TYPE ST_ProbesSettings :
STRUCT
	
	anDistanceCalibrationBlock			: ARRAY [1..3] OF REAL;	
	nDistanceOffset1					: ARRAY [1..3] OF REAL; 
	nDistanceOffset2					: ARRAY [1..3] OF REAL;
	(*Renan Added 30Jun26 - Nests offset*)
	anNestOffsetByProbe1         		: ARRAY [1..4] OF REAL;
    anNestOffsetByProbe2         		: ARRAY [1..4] OF REAL;
	(*/Renan Added 30Jun26*)	
	anExpectedDistances					: ARRAY [1..3] OF REAL;
	anHeightSetByCalibration1			: ARRAY [1..4] OF REAL;	
	anHeightSetByCalibration2			: ARRAY [1..4] OF REAL;	
	anTolerances						: ARRAY [1..3] OF REAL;	


END_STRUCT
END_TYPE

(* stored: Version 1.1.0.1, ProductVersion 3.1.4026.18
   DUT ST_ProbesSettings: Id {a88f077e-6c66-4a83-be94-fdfa4e9dc786} *)
